(* CODESYS project EmiconSys.library
   Author: Emicon
   Placeholder: EmiconSys
   Title: Emicon system functions
   Version: 3.5.13.0
   DefaultNamespace: EMSys
   Company: Emicon

Project tree, tasks and I/O mapping:
  libraries: CmpApp, * (System); CmpEventMgr, * (System); Standard, * (System); SysFile, * (System); SysTypes Interfaces, * (System); SysCom, * (System); SysMem, * (System)
  function block EventHandler [ST]: xDenyOperation, EventCallback, FB_Init, FB_Exit
  function set_inhibit [ST]
  function set_watchdog [ST]
  function Get_ptr_to_DPM [ST]
  function Get_ptr_to_slot0 [ST]
  function PUTS [ST]
  function SysSync [ST]
  function Get_ptr_to_sock_arr [ST]
  global variables GVL
  function block FreeAllMem [ST]: FB_Exit, FB_Init
  function MemAlloc [ST]
  function MemFree [ST]
  function MemRealloc [ST]
*)

// GVL
{attribute 'hide'}
VAR_GLOBAL CONSTANT
	BuffPtrZize			: UINT	:=2048;
END_VAR
VAR_GLOBAL
	InitDisplPortFlag	: BOOL;
	hCom 				: RTS_IEC_HANDLE;
	BuffMemPtr			: POINTER TO POINTER TO BYTE;
	FAM					: FreeAllMem;
END_VAR

// EventHandler
{attribute 'm4export_hide'}
{attribute 'hide'}
FUNCTION_BLOCK EventHandler IMPLEMENTS ICmpEventCallback
VAR_INPUT
END_VAR
VAR_OUTPUT
END_VAR
VAR
	_dwEventId:			DWORD;
	_hEvent:			RTS_IEC_HANDLE;
	_hCallbackHandler:	RTS_IEC_HANDLE;	
	_xDeny : BOOL;
END_VAR

PROPERTY xDenyOperation : bool
SET
_xDeny := xDenyOperation;
END_SET
GET
xDenyOperation := _xDeny;
END_GET
END_PROPERTY

{attribute 'm4export_hide'}
{attribute '''NORMAL__COMMENT' := ' The interface ICmpEventCallback must be registered for an event. If this event is posted, this callback method is called.'}

(* The interface ICmpEventCallback must be registered for an event. If this event is posted, this callback method is called.*)
METHOD EventCallback : CmpEventMgr.RTS_IEC_RESULT
VAR_INPUT
	(*Pointer to the event parameters, see Struct EventParam*)
	pEventParam	: POINTER TO CmpEventMgr.EventParam;
	//EventPrm : CmpApp.EVTPARAM_CmpApp;
END_VAR
VAR
	pEventParamDenyStop:	POINTER TO EVTPARAM_CmpAppDenyStop;
	pParam : POINTER TO EVTPARAM_CmpApp;
	udiState : UDINT;
	hFile : RTS_IEC_HANDLE;
	str_value: STRING[2];
	fileResult : UDINT;
END_VAR
pParam := pEventParam^.pParameter;
udiState := pParam^.pApp^.udiState;
						
//GVL.count := udiState;

IF udiState = 1 THEN
	str_value := '0';	
ELSE
	str_value := '1';
END_IF

hFile := SysFileOpen('/sys/class/gpio/gpio96/value', AM_WRITE ,ADR(fileResult));
SysFileWrite(hFile, ADR(str_value),  INT_TO_DWORD(len(str_value)), ADR(fileResult));
SysFileClose(hFile);
END_METHOD

METHOD FB_Init
VAR_INPUT
	bInitRetains: BOOL;     
	bInCopyCode: BOOL;	
	dwEventId:		DWORD;
END_VAR
VAR
	result:	RTS_IEC_RESULT;
END_VAR
_dwEventId := dwEventId;
_xDeny := FALSE;

_hEvent := EventOpen( dwEventId , CmpApp.CMPID_CmpApp, result );

_hCallbackHandler := EventRegisterCallback(_hEvent, THIS^ , result );
END_METHOD

METHOD FB_Exit : RTS_IEC_RESULT
VAR_INPUT
	bInCopyCode: BOOL;
END_VAR
IF _hCallbackHandler <> CmpEventMgr.RTS_INVALID_HANDLE THEN
	EventUnregisterCallback( _dwEventId, _hCallbackHandler );
END_IF

IF _hEvent <> CmpEventMgr.RTS_INVALID_HANDLE THEN
	EventClose2( _hEvent );	 
END_IF
END_METHOD

END_FUNCTION_BLOCK

// set_inhibit
{attribute 'hide'}
FUNCTION set_inhibit : int
VAR_INPUT
END_VAR
VAR
END_VAR

END_FUNCTION

// set_watchdog
{attribute 'hide'}
FUNCTION set_watchdog : int
VAR_INPUT
END_VAR
VAR
END_VAR

END_FUNCTION

// Get_ptr_to_DPM
{attribute 'hide'}
FUNCTION Get_ptr_to_DPM : POINTER TO WORD
VAR_INPUT
END_VAR
VAR
END_VAR

(*********************************************************)
(*  ЛУЧИН Е.В.                                           *)
(*  07.07.2016                                           *)
(*  Функция возвращает указатель на начало виртуальной   *)
(*  памяти куда мапирется адресное пространство ДПМ      *)
(*********************************************************)

END_FUNCTION

// Get_ptr_to_slot0
{attribute 'hide'}
FUNCTION Get_ptr_to_slot0 : POINTER TO BYTE
VAR_INPUT
END_VAR
VAR
END_VAR

(*********************************************************)
(*  ЛУЧИН Е.В.                                           *)
(*  07.07.2016                                           *)
(*  Функция возвращает указатель на начало виртуальной   *)
(*  памяти куда мапирется адресное пространство слотов   *)
(*********************************************************)

END_FUNCTION

// PUTS
{attribute 'm4export_hide'}
{attribute 'hide'}
FUNCTION PUTS: INT
VAR_INPUT
	iLine: INT;		// Строка 0-1
	iPos: INT;		// Столбец 0-249
	stData: STRING;	// Текст 1-250 сиволов
END_VAR
VAR
	buff: ARRAY[0..255] OF BYTE;
	buff_len: INT;
	str_len: INT;
	i:INT;
	result : RTS_IEC_RESULT;
	csComSettings: COM_Settings;	
END_VAR

(*********************************************************)
(*  company:  ЗАО "ЭМИКОН"                               *)
(*  author:   ЛУЧИН Е.В.                                 *)
(*  date of last modification:  14.03.2017               *)
(*  description:                                         *)
(*  Функция для вывода строк на дисплей                  *)
(*********************************************************)
   
PUTS:=0;
IF iLine > 1 THEN RETURN; END_IF
IF iLine < 0 THEN RETURN; END_IF
IF iPos > 249 THEN RETURN; END_IF
IF iPos < 0 THEN RETURN; END_IF

str_len:=LEN(stData);
IF str_len > 250 THEN str_len:=250;	END_IF

buff[0]:=INT_TO_BYTE(iPos);
buff[1]:=INT_TO_BYTE(iLine);

FOR i:= 0 TO str_len DO
	buff[i+2]:=stData[i];
END_FOR
buff[i+1]:=16#FF;

IF NOT InitDisplPortFlag THEN
	hCom := SysComOpen(sPort:= SYS_COMPORT3 , pResult:= ADR(result));
	IF hCom <> RTS_INVALID_HANDLE THEN
		// Configure the connection
		csComSettings.byParity := SysCom.SYS_EVENPARITY;
		csComSettings.byStopBits := SysCom.SYS_TWOSTOPBITS;
		csComSettings.sPort := SYS_COMPORT3;
		csComSettings.ulBaudrate := SysCom.SYS_BR_57600;
		csComSettings.ulBufferSize := 0;
		csComSettings.ulTimeout := 0; //10
		Result := SysComSetSettings(hCom:= hCom, pSettings:= ADR(csComSettings), pSettingsEx:= 0);
		InitDisplPortFlag:= TRUE;		
	ELSE
		PUTS:=0;
		RETURN;
	END_IF
END_IF

IF hCom <> RTS_INVALID_HANDLE THEN
	SysComWrite(hCom:= hCom,
				pbyBuffer:= ADR(buff),
				ulSize:= INT_TO_UDINT(str_len+3),
				ulTimeout:= 50,//100
				pResult:= ADR(result));
ELSE
	PUTS:=0;
	InitDisplPortFlag:=FALSE;
	RETURN;	
END_IF

PUTS:=str_len+iPos;
IF PUTS > 250 THEN PUTS:=0; END_IF

END_FUNCTION

// SysSync
FUNCTION SysSync : INT
VAR_INPUT
END_VAR
VAR
END_VAR

END_FUNCTION

// Get_ptr_to_sock_arr
{attribute 'hide'}
FUNCTION Get_ptr_to_sock_arr : pointer to udint
VAR_INPUT
END_VAR
VAR
END_VAR

END_FUNCTION

// FreeAllMem
{attribute 'm4export_hide'}
{attribute 'hide'}
FUNCTION_BLOCK FreeAllMem
VAR_INPUT
END_VAR
VAR_OUTPUT
END_VAR
VAR
END_VAR

METHOD FB_Exit : BOOL
VAR_INPUT
	bInCopyCode: BOOL;
END_VAR
END_METHOD

METHOD  FB_Init : BOOL
VAR_INPUT
	bInitRetains: BOOL;
	bInCopyCode: BOOL;	
END_VAR
VAR 
	i	: UINT;
	BP	: POINTER TO POINTER TO BYTE;
	rez	: RTS_IEC_RESULT;
END_VAR
(*********************************************************)
(*  company:  ЗАО "ЭМИКОН"                               *)
(*  author:   ЛУЧИН Е.В.                                 *)
(*  date of last modification:  19.04.2018               *)
(*  description:                                         *)
(*  Метод для автоматического освобождения динамической  *)
(*  памяти при старте проекта      		                 *)
(*********************************************************)
BP:=Get_ptr_to_sock_arr();	// получаю указатель на скрытое хранилище
IF BP > 0 THEN				// при успешном получении указателя
	BuffMemPtr:=BP[255];	// получаю указатель на буфер зачистки
	IF BuffMemPtr > 0 THEN	// при наличии буфера
		FOR i:=0 TO BuffPtrZize - 1 DO	// обхожу буфер для освобождения ранее выделенной памяти
			IF BuffMemPtr[i] > 0 THEN
				SysMemFreeData(	szComponent:='EMSYS' , 
								pMemory:=BuffMemPtr[i] );
				BuffMemPtr[i]:=0;
			END_IF
		END_FOR
		
	ELSE					// если буфер зачистки не существует
		BuffMemPtr:=SysMemAllocData(szComponent:='EMSYS' , // то создаю его
									udiSize:=BuffPtrZize*SIZEOF(POINTER TO BYTE) , 
									pResult:=ADR(rez) );
		BP[255]:=BuffMemPtr;	// и сохраняю указатель на буфер в скрытом хранилище
		IF BuffMemPtr > 0 THEN	// зануляю содержимое буфера
			FOR i:=0 TO BuffPtrZize - 1 DO
				BuffMemPtr[i]:=0;
			END_FOR			
		END_IF
	END_IF
	
ELSE
	BuffMemPtr:=0;
END_IF
END_METHOD

END_FUNCTION_BLOCK

// MemAlloc
(*
Функция для динамического выделения памяти
*)
FUNCTION MemAlloc : pointer to byte
VAR_INPUT
	udiSize	: UDINT; // размер запрашиваемого блока памяти
END_VAR
VAR
	i	: UINT;
	rez	: RTS_IEC_RESULT;
END_VAR

(*********************************************************)
(*  company:  ЗАО "ЭМИКОН"                               *)
(*  author:   ЛУЧИН Е.В.                                 *)
(*  date of last modification:  19.04.2018               *)
(*  description:                                         *)
(*  Функция для динамического выделения памяти   	     *)
(*                              		                 *)
(*********************************************************)

MemAlloc:=SysMemAllocData(szComponent:='EMSYS' , udiSize:=udiSize , pResult:=ADR(rez) ); // выделяю память

IF MemAlloc > 0 
AND BuffMemPtr > 0 THEN					// заношу указатель в буфер зачистки при успешном выделении памяти
	FOR i:=0 TO BuffPtrZize - 1 DO
		IF BuffMemPtr[i] = 0 THEN
			BuffMemPtr[i]:=MemAlloc;
			RETURN;
		END_IF
	END_FOR
END_IF

END_FUNCTION

// MemFree
(*
Функция для освобождения динамически выделенной памяти
*)
FUNCTION MemFree : BOOL
VAR_INPUT
	pbyPtr	: POINTER TO BYTE; // Указатель на блок выделенной памяти
END_VAR
VAR
	i	: uint;
END_VAR

(*********************************************************)
(*  company:  ЗАО "ЭМИКОН"                               *)
(*  author:   ЛУЧИН Е.В.                                 *)
(*  date of last modification:  19.04.2018               *)
(*  description:                                         *)
(*  Функция для освобождения            			     *)
(*  динамически выделенной памяти		                 *)
(*********************************************************)
IF pbyPtr = 0 THEN
	RETURN;
END_IF

SysMemFreeData(szComponent:='EMSYS' , pMemory:=pbyPtr ); // освобождаю память
IF BuffMemPtr > 0 THEN
	FOR i:=0 TO BuffPtrZize - 1 DO		// убираю указатель из буфера зачистки
		IF BuffMemPtr[i] = pbyPtr THEN
			BuffMemPtr[i]:=0;
			RETURN;
		END_IF
	END_FOR	
END_IF

END_FUNCTION

// MemRealloc
(*
Функция для изменения размера ранее выделенного блока динамической памяти 
*)
FUNCTION MemRealloc : POINTER TO BYTE
VAR_INPUT
	pbyPtr	: POINTER TO BYTE; 	// указатель на ранее выделенный блок памяти
	udiSize	: UDINT;			// новый размер блока памяти
END_VAR
VAR
	i	: UINT;
	rez	: RTS_IEC_RESULT;
END_VAR

(*********************************************************)
(*  company:  ЗАО "ЭМИКОН"                               *)
(*  author:   ЛУЧИН Е.В.                                 *)
(*  date of last modification:  19.04.2018               *)
(*  description:                                         *)
(*  Функция для изменения размера ранее выделенного      *)
(*  блока динамической памяти          	                 *)
(*********************************************************)

IF pbyPtr > 0 THEN // если есть входной указатель
	MemRealloc:=SysMemReallocData(	szComponent:='EMSYS' , // изменяю размер ранее выделенного блока памяти
									pMemory:=pbyPtr , 
									udiSize:=udiSize , 
									pResult:=ADR(rez) );	
	IF MemRealloc <> pbyPtr 
	AND BuffMemPtr > 0THEN							// если поменялся указатель на блок памяти
		FOR i:=0 TO BuffPtrZize - 1 DO						// меняю его в буфере зачистки
			IF BuffMemPtr[i] = pbyPtr THEN
				BuffMemPtr[i]:=MemRealloc;
				RETURN;
			END_IF
		END_FOR		
	END_IF
	
ELSE														// при отсутствии входного указателя
	MemRealloc:=SysMemAllocData(szComponent:='EMSYS' , 
								udiSize:=udiSize , 
								pResult:=ADR(rez) ); // выделяю память
	IF MemRealloc > 0 
	AND BuffMemPtr > 0 THEN					// заношу указатель в буфер зачистки
		FOR i:=0 TO BuffPtrZize - 1 DO
			IF BuffMemPtr[i] = 0 THEN
				BuffMemPtr[i]:=MemRealloc;
				RETURN;
			END_IF
		END_FOR
	END_IF	
END_IF

END_FUNCTION
